TYPE TimeInfo :
STRUCT
	dctime: T_DCTIME64; (* The DC time gotten from F_GetActualDcTime64(). *)
    dctotcoff: LINT; (* Offset between DC and TwinCAT time (in ns). *)
	dctoextoff: LINT; (* Offset between DC and external time (in ns). *)
	internalstamp: ULINT; (* Internal timestamp from EL6688. *)
	externalstamp: ULINT; (* External timestamp from EL6688. *)
END_STRUCT
END_TYPE

(* stored: Version 1.1.0.1, ProductVersion 3.1.4022.12
   DUT TimeInfo: Id {6fb7af14-518c-40e5-95d9-d3ee85114f02} *)
